{attribute addProperty BoxType "EL3773-0000-0016"}
{attribute addProperty Id "UnderrangeBIT10.1251OverrangeBIT10.1252Limit_1_BIT_0BIT10.1253Limit_1_BIT_1BIT10.1253Limit_2_BIT_0BIT10.1255Limit_2_BIT_1BIT10.1255ErrorBIT10.1257Sync_errorBIT10.12532TxPDO_StateBIT10.1257TxPDO_ToggleBIT10.1259"}
{attribute addProperty CRC "4189364243"}
{attribute addProperty SizeInBites "16"}
{attribute addProperty SizeInBytes "2"}
TYPE I1_STATUS_F9B4A013 :
STRUCT
	{attribute addProperty Name "Underrange"}
	Underrange : BIT;
	{attribute addProperty Name "Overrange"}
	Overrange : BIT;
	{attribute addProperty Name "Limit_1"}
	Limit_1_BIT_0 : BIT;
	{attribute addProperty Name "Limit_1"}
	Limit_1_BIT_1 : BIT;
	{attribute addProperty Name "Limit_2"}
	Limit_2_BIT_0 : BIT;
	{attribute addProperty Name "Limit_2"}
	Limit_2_BIT_1 : BIT;
	{attribute addProperty Name "Error"}
	Error : BIT;
	{attribute 'hide'}
	reserve_1 : BIT;
	{attribute 'hide'}
	reserve_2_BIT_0 : BIT;
	{attribute 'hide'}
	reserve_2_BIT_1 : BIT;
	{attribute 'hide'}
	reserve_2_BIT_2 : BIT;
	{attribute 'hide'}
	reserve_2_BIT_3 : BIT;
	{attribute 'hide'}
	reserve_2_BIT_4 : BIT;
	{attribute addProperty Name "Sync_error"}
	Sync_error : BIT;
	{attribute addProperty Name "TxPDO_State"}
	TxPDO_State : BIT;
	{attribute addProperty Name "TxPDO_Toggle"}
	TxPDO_Toggle : BIT;
END_STRUCT
END_TYPE

(* stored: Version 1.2.0.0, ProductVersion 3.1.4024.9
   DUT I1_STATUS_F9B4A013: Id {7a291e27-91c1-456f-9982-5473e70b3c10} *)
